FOR i := 0 TO (_Count - 1) DO
	IF _Data[i] = Item THEN
		_Data[i]	 := 0;
		removedItems := removedItems + 1;
	END_IF
END_FOR

IF _Count > 1 THEN
	FOR i := 0 TO (_Count - 2) DO
		IF _Data[i] = 0 AND _Data[i + 1] <> 0 THEN
			_Data[i]	 := _Data[i + 1];
			_Data[i + 1] := 0;
		END_IF
	END_FOR
END_IF

CountListItems();
_Count := _Count - removedItems;
END_METHOD

END_FUNCTION_BLOCK

// ---- _Internal/MotionTasks/MC2/AX5000/Mc2MotionTask_AX5000AmpToNm.TcPOU
FUNCTION_BLOCK Mc2MotionTask_AX5000AmpToNm EXTENDS Mc2MotionTask
VAR
	i					   : INT;
	SequenceState		   : DINT := -10;
	RawConfigChPeakCurrent : UDINT;					// Configured Channel Peak Current  ( raw )
	ConfigChPeakCurrent	   : LREAL;					// Configured Channel Peak Current  ( units := A )
	MotorConsType		   : WORD;					// Motor construction type          ( raw )
	MotorType			   : BOOL;					// Motor construction type          ( units := 0 = Rotary, 1 = Linear ) 
	RawContStallTorque	   : UDINT;					// Motor continuous stall torque    ( raw )
	ContStallTorque		   : LREAL;					// Motor continuous stall torque    ( units := Nm )
	ContStallTorqueEx	   : LREAL;					// Motor continuous stall torque    ( units := Nm ) - extended slope   
	RawPeakTorque		   : UDINT;					// Motor peak torque                ( raw )
	PeakTorque			   : LREAL;					// Motor peak torque                ( units := Nm )
	RawContStallForce	   : UDINT;					// Motor continuous stall force     ( raw )
	ContStallForce		   : LREAL;					// Motor continuous stall force     ( units := N )
	ContStallForceEx	   : LREAL;					// Motor continuous stall force     ( units := N ) - extended slope
	RawPeakForce		   : UDINT;					// Motor peak force                 ( raw )
	PeakForce			   : LREAL;					// Motor peak force                 ( units := N )
	RawContStallCurrent	   : UDINT;					// Motor continuous stall current   ( raw )
	ContStallCurrent	   : LREAL;					// Motor continuous stall current   ( units := A )
	ContStallCurrentEx	   : LREAL;					// Motor continuous stall current   ( units := A ) - extended slope
	RawPeakCurrent		   : UDINT;					// Motor peak current               ( raw )
	PeakCurrent			   : LREAL;					// Motor peak current               ( units := A )
	Scale				   : LREAL;					// Position between array indexes   ( units := % )
	SoERead				   : FB_SoERead;			// Read SoE params from drive
	RawMotorTorqueCurve	   : ST_IDN_P_0_0074_UDINT; // Contents read in from P-0-0074   ( raw )
END_VAR

VAR
	_ErrorId		 : UDINT;			 // 1 = Axis Not Linked, 2 = Failed To Read P-0-0074, 3 = Failed To Read P-0-0092, 4 = Failed To Read P-0-0050, 5 = Failed To Read P-0-0070, 6 = Failed To Read P-0-0126, 7 = Failed To Read S-0-0111
	CalculatedValues : ST_AX5000AmpToNm; // Data read in and calculated from the drive
END_VAR

(*  
Error Ids:
  1 = Axis Not Linked, 
  2 = Failed To Read P-0-0074,
  3 = Failed To Read P-0-0092, 
  4 = Failed To Read P-0-0050, 
  5 = Failed To Read P-0-0070, 
  6 = Failed To Read P-0-0126, 
  7 = Failed To Read S-0-0111 
*)

{attribute 'monitoring' := 'call'}
PROPERTY ActCurrent : LREAL
GET
ActCurrent := CalculatedValues.ActCurrent;
END_GET
END_PROPERTY

{attribute 'monitoring' := 'call'}
PROPERTY ActTorque : LREAL
GET
ActTorque := CalculatedValues.ActTorque;
END_GET
END_PROPERTY

{attribute 'monitoring' := 'call'}
PROPERTY Busy : BOOL
GET
Busy := SequenceState > 0 AND SequenceState <= 100;
END_GET
END_PROPERTY

METHOD CyclicLogic
IF _Axis = 0 THEN
	RETURN;
END_IF

CASE SequenceState OF
	-10: // Initialize
		RawConfigChPeakCurrent := 0;
		ConfigChPeakCurrent	   := 0.0;
		MotorConsType		   := 0;
		MotorType			   := FALSE;
		RawContStallTorque	   := 0;
		ContStallTorque		   := 0.0;
		ContStallTorqueEx	   := 0.0;
		RawPeakTorque		   := 0;
		PeakTorque			   := 0.0;
		RawContStallForce	   := 0;
		ContStallForce		   := 0.0;
		ContStallForceEx	   := 0.0;
		RawPeakForce		   := 0;
		PeakForce			   := 0.0;
		RawContStallCurrent	   := 0;
		ContStallCurrent	   := 0.0;
		ContStallCurrentEx	   := 0.0;
		RawPeakCurrent		   := 0;
		PeakCurrent			   := 0.0;
		Scale				   := 0.0;
		SoERead(Execute := FALSE, Axis := _Axis.Axis);
		MEMSET(ADR(RawMotorTorqueCurve), 16#0, SIZEOF(RawMotorTorqueCurve));
		MEMSET(ADR(CalculatedValues), 16#0, SIZEOF(CalculatedValues));
		IF _Axis.Axis.NcToPlc.AxisId = 0 THEN
			_ErrorId	  := 1;
			SequenceState := 5000;
		ELSE
			SequenceState := SequenceState + 10;
		END_IF

	0:	// Wait for Execute()  
	10: // Read in the value of P-0-0074 ( Motor torque characteristic )
		SoERead(NetId	:= '',
				Idn		:= P_0_IDNs + 74,
				Element := 16#40,
				pDstBuf := ADR(RawMotorTorqueCurve),
				BufLen	:= SIZEOF(RawMotorTorqueCurve),
				Execute := TRUE,
				Axis	:= _Axis.Axis);

		IF NOT SoERead.Busy AND NOT SoERead.Error THEN
			SoERead(Execute := FALSE, Axis := _Axis.Axis);
			FOR i := 0 TO 9 DO // Convert raw values into actual units
				CalculatedValues.Curve.Iq[i] := UDINT_TO_LREAL(RawMotorTorqueCurve.Elements.Iq[i]) / 1000.0;
				CalculatedValues.Curve.M[i]	 := UDINT_TO_LREAL(RawMotorTorqueCurve.Elements.M[i]) / 100.0;
			END_FOR

			SequenceState := SequenceState + 10;
		ELSIF SoERead.Error THEN
			SoERead(Execute := FALSE, Axis := _Axis.Axis);
			_ErrorId	  := 2;
			SequenceState := 5000;
		END_IF

	20: // Read in the value of P-0-0092 ( Configured channel peak current )       
		SoERead(NetId	:= '',
				Idn		:= P_0_IDNs + 92,
				Element := 16#40,
				pDstBuf := ADR(RawConfigChPeakCurrent),
				BufLen	:= SIZEOF(RawConfigChPeakCurrent),
				Execute := TRUE,
				Axis	:= _Axis.Axis);

		IF NOT SoERead.Busy AND NOT SoERead.Error THEN // Convert raw values into actual units
			SoERead(Execute := FALSE, Axis := _Axis.Axis);
			ConfigChPeakCurrent := UDINT_TO_LREAL(RawConfigChPeakCurrent) / 1000.0;
			SequenceState		:= SequenceState + 10;
		ELSIF SoERead.Error THEN
			SoERead(Execute := FALSE, Axis := _Axis.Axis);
			_ErrorId	  := 3;
			SequenceState := 5000;
		END_IF

	30: // Check for valid characteristic curve
		IF RawMotorTorqueCurve.Elements.Iq[9] = 0 THEN
			SequenceState := SequenceState + 10; // Curve is not available
		ELSE
			SequenceState := 1000; // Curve is available
		END_IF

	40: // Read in the value of P-0-0050 ( Motor construction type )       
		SoERead(NetId	:= '',
				Idn		:= P_0_IDNs + 50,
				Element := 16#40,
				pDstBuf := ADR(MotorConsType),
				BufLen	:= SIZEOF(MotorConsType),
				Execute := TRUE,
				Axis	:= _Axis.Axis);

		IF NOT SoERead.Busy AND NOT SoERead.Error THEN
			SoERead(Execute := FALSE, Axis := _Axis.Axis);
			MotorType := MotorConsType.1;
			IF NOT MotorType THEN
				SequenceState := 50; // Rotary
			ELSE
				SequenceState := 70; // Linear
			END_IF
		ELSIF SoERead.Error THEN
			SoERead(Execute := FALSE, Axis := _Axis.Axis);
			_ErrorId	  := 4;
			SequenceState := 5000;
		END_IF

	50: // Read in the value of P-0-0070 ( Motor continuous stall torque )       
		SoERead(NetId	:= '',
				Idn		:= P_0_IDNs + 70,
				Element := 16#40,
				pDstBuf := ADR(RawContStallTorque),
				BufLen	:= SIZEOF(RawContStallTorque),
				Execute := TRUE,
				Axis	:= _Axis.Axis);

		IF NOT SoERead.Busy AND NOT SoERead.Error THEN
			SoERead(Execute := FALSE, Axis := _Axis.Axis);
			ContStallTorque := UDINT_TO_LREAL(RawContStallTorque) / 100.0;
			SequenceState	:= SequenceState + 10;
		ELSIF SoERead.Error THEN
			SoERead(Execute := FALSE, Axis := _Axis.Axis);
			_ErrorId	  := 5;
			SequenceState := 5000;
		END_IF

	60: // Read in the value of P-0-0073 ( Motor peak torque )       
		SoERead(NetId	:= '',
				Idn		:= P_0_IDNs + 73,
				Element := 16#40,
				pDstBuf := ADR(RawPeakTorque),
				BufLen	:= SIZEOF(RawPeakTorque),
				Execute := TRUE,
				Axis	:= _Axis.Axis);

		IF NOT SoERead.Busy AND NOT SoERead.Error THEN
			SoERead(Execute := FALSE, Axis := _Axis.Axis);
			PeakTorque	  := UDINT_TO_LREAL(RawPeakTorque) / 100.0;
			SequenceState := 90;
		ELSIF SoERead.Error THEN
			SoERead(Execute := FALSE, Axis := _Axis.Axis);
			SequenceState := 90;
		END_IF

	70: // Read in the value of P-0-0126 ( Motor continuous stall force )       
		SoERead(NetId	:= '',
				Idn		:= P_0_IDNs + 126,
				Element := 16#40,
				pDstBuf := ADR(RawContStallForce),
				BufLen	:= SIZEOF(RawContStallForce),
				Execute := TRUE,
				Axis	:= _Axis.Axis);

		IF NOT SoERead.Busy AND NOT SoERead.Error THEN
			SoERead(Execute := FALSE, Axis := _Axis.Axis);
			ContStallForce := UDINT_TO_LREAL(RawContStallForce) / 100.0;
			SequenceState  := SequenceState + 10;
		ELSIF SoERead.Error THEN
			SoERead(Execute := FALSE, Axis := _Axis.Axis);
			_ErrorId	  := 6;
			SequenceState := 5000;
		END_IF

	80: // Read in the value of P-0-0128 ( Motor peak force )       
		SoERead(NetId	:= '',
				Idn		:= P_0_IDNs + 128,
				Element := 16#40,
				pDstBuf := ADR(RawPeakForce),
				BufLen	:= SIZEOF(RawPeakForce),
				Execute := TRUE,
				Axis	:= _Axis.Axis);

		IF NOT SoERead.Busy AND NOT SoERead.Error THEN
			SoERead(Execute := FALSE, Axis := _Axis.Axis);
			PeakForce	  := UDINT_TO_LREAL(RawPeakForce) / 100.0;
			SequenceState := SequenceState + 10;
		ELSIF SoERead.Error THEN
			SoERead(Execute := FALSE, Axis := _Axis.Axis);
			SequenceState := SequenceState + 10;
		END_IF

	90: // Read in the value of S-0-0111 ( Motor continuous stall current )       
		SoERead(NetId	:= '',
				Idn		:= S_0_IDNs + 111,
				Element := 16#40,
				pDstBuf := ADR(RawContStallCurrent),
				BufLen	:= SIZEOF(RawContStallCurrent),
				Execute := TRUE,
				Axis	:= _Axis.Axis);

		IF NOT SoERead.Busy AND NOT SoERead.Error THEN
			SoERead(Execute := FALSE, Axis := _Axis.Axis);
			ContStallCurrent := UDINT_TO_LREAL(RawContStallCurrent) / 1000.0;
			SequenceState	 := SequenceState + 10;
		ELSIF SoERead.Error THEN
			SoERead(Execute := FALSE, Axis := _Axis.Axis);
			_ErrorId	  := 7;
			SequenceState := 5000;
		END_IF

	100: // Read in the value of S-0-0109 ( Motor peak current )       
		SoERead(NetId	:= '',
				Idn		:= S_0_IDNs + 109,
				Element := 16#40,
				pDstBuf := ADR(RawPeakCurrent),
				BufLen	:= SIZEOF(RawPeakCurrent),
				Execute := TRUE,
				Axis	:= _Axis.Axis);

		IF NOT SoERead.Busy THEN
			SoERead(Execute := FALSE, Axis := _Axis.Axis);
			PeakCurrent := UDINT_TO_LREAL(RawPeakCurrent) / 1000.0;
			IF NOT MotorType THEN
				IF PeakCurrent = 0 OR PeakTorque = 0 THEN
					SequenceState := 300; // Rotary Motor: Curve not available... peak torque and current missing - Using slope of points 0,0 to P-0-0070 and S-0-0111
				ELSE
					SequenceState := 200; // Rotary Motor: Curve not available - Using linear interpolation of points P-0-0070, P-0-0073, S-0-0111 and S-0-0109
				END_IF
			ELSE
				IF PeakCurrent = 0 OR PeakForce = 0 THEN
					SequenceState := 500; // Linear Motor: Curve not available... peak torque and current missing - Using slope of points 0,0 to P-0-0126 and S-0-0111
				ELSE
					SequenceState := 400; // Linear Motor: Curve not available - Using linear interpolation of points P-0-0126, P-0-0128, S-0-0111 and S-0-0109
				END_IF
			END_IF
		END_IF

	200: // Rotary Motor: Curve not available - Using linear interpolation of points P-0-0070, P-0-0073, S-0-0111 and S-0-0109
		CalculatedValues.ActCurrent := ABS((_Axis.Axis.NcToPlc.ActTorque / 100) * ConfigChPeakCurrent);
		// Convert the actual current in amps to Nm
		IF CalculatedValues.ActCurrent = 0 THEN
			CalculatedValues.ActTorque := 0;
		ELSIF CalculatedValues.ActCurrent > 0 AND CalculatedValues.ActCurrent < ContStallCurrent THEN
			IF ContStallCurrent > 0 THEN
				Scale					   := CalculatedValues.ActCurrent / ContStallCurrent;
				CalculatedValues.ActTorque := Scale * ContStallTorque;
			END_IF
		ELSIF CalculatedValues.ActCurrent >= ContStallCurrent AND CalculatedValues.ActCurrent <= PeakCurrent THEN
			IF (CalculatedValues.ActCurrent - ContStallCurrent) > 0 AND (PeakCurrent - ContStallCurrent) > 0 THEN
				Scale					   := (CalculatedValues.ActCurrent - ContStallCurrent) / (PeakCurrent - ContStallCurrent);
				CalculatedValues.ActTorque := (Scale * (PeakTorque - ContStallTorque) + ContStallTorque);
			END_IF
		END_IF

	300: // Rotary Motor: Curve not available... peak torque and current missing - Using slope of points 0,0 to P-0-0070 and S-0-0111
		CalculatedValues.ActCurrent := ABS((_Axis.Axis.NcToPlc.ActTorque / 100) * ConfigChPeakCurrent);

		// Project slope from continuous stall torque/current
		ContStallCurrentEx := ContStallCurrent * 10.0;
		ContStallTorqueEx  := ContStallTorque * 10.0;
		// Convert the actual current in amps to Nm
		IF CalculatedValues.ActCurrent = 0 THEN
			CalculatedValues.ActTorque := 0;
		ELSIF CalculatedValues.ActCurrent > 0 AND CalculatedValues.ActCurrent <= ContStallCurrentEx THEN
			IF ContStallCurrentEx > 0 THEN
				Scale					   := CalculatedValues.ActCurrent / ContStallCurrentEx;
				CalculatedValues.ActTorque := Scale * ContStallTorqueEx;
			END_IF
		END_IF

	400: // Linear Motor: Curve not available - Using linear interpolation of points P-0-0126, P-0-0128, S-0-0111 and S-0-0109
		CalculatedValues.ActCurrent := ABS((_Axis.Axis.NcToPlc.ActTorque / 100) * ConfigChPeakCurrent);
		// Convert the actual current in amps to Nm
		IF CalculatedValues.ActCurrent = 0 THEN
			CalculatedValues.ActTorque := 0;
		ELSIF CalculatedValues.ActCurrent > 0 AND CalculatedValues.ActCurrent < ContStallCurrent THEN
			IF ContStallCurrent > 0 THEN
				Scale					   := CalculatedValues.ActCurrent / ContStallCurrent;
				CalculatedValues.ActTorque := Scale * ContStallForce;
			END_IF
		ELSIF CalculatedValues.ActCurrent >= ContStallCurrent AND CalculatedValues.ActCurrent <= PeakCurrent THEN
			IF (CalculatedValues.ActCurrent - ContStallCurrent) > 0 AND (PeakCurrent - ContStallCurrent) > 0 THEN
				Scale					   := (CalculatedValues.ActCurrent - ContStallCurrent) / (PeakCurrent - ContStallCurrent);
				CalculatedValues.ActTorque := (Scale * (PeakForce - ContStallForce) + ContStallForce);
			END_IF
		END_IF

	500: // Linear Motor: Curve not available... peak torque and current missing - Using slope of points 0,0 to P-0-0126 and S-0-0111
		CalculatedValues.ActCurrent := ABS((_Axis.Axis.NcToPlc.ActTorque / 100) * ConfigChPeakCurrent);

		// Project slope from continuous stall torque/current
		ContStallCurrentEx := ContStallCurrent * 10.0;
		ContStallForceEx   := ContStallForce * 10.0;
		// Convert the actual current in amps to Nm
		IF CalculatedValues.ActCurrent = 0 THEN
			CalculatedValues.ActTorque := 0;
		ELSIF CalculatedValues.ActCurrent > 0 AND CalculatedValues.ActCurrent <= ContStallCurrentEx THEN
			IF ContStallCurrentEx > 0 THEN
				Scale					   := CalculatedValues.ActCurrent / ContStallCurrentEx;
				CalculatedValues.ActTorque := Scale * ContStallForceEx;
			END_IF
		END_IF

	1000: // Rotary or Linear Motor: Curve available - Compare actual torque value in Amps to the characteristic curve and output actual torque value in Nm
		CalculatedValues.ActCurrent := ABS((_Axis.Axis.NcToPlc.ActTorque / 100) * ConfigChPeakCurrent);
		// Convert the actual current in amps to Nm
		FOR i := 1 TO 9 DO
			IF CalculatedValues.ActCurrent = 0 THEN
				CalculatedValues.ActTorque := 0;
				EXIT;
			ELSIF CalculatedValues.ActCurrent > 0 AND CalculatedValues.ActCurrent < CalculatedValues.Curve.Iq[0] THEN
				IF CalculatedValues.Curve.Iq[0] > 0 THEN
					Scale					   := CalculatedValues.ActCurrent / CalculatedValues.Curve.Iq[0];
					CalculatedValues.ActTorque := Scale * CalculatedValues.Curve.M[0];
				END_IF

				EXIT;
			ELSIF CalculatedValues.ActCurrent >= CalculatedValues.Curve.Iq[i - 1] AND CalculatedValues.ActCurrent <= CalculatedValues.Curve.Iq[i] THEN
				IF (CalculatedValues.Curve.Iq[i] - CalculatedValues.Curve.Iq[i - 1]) > 0 AND CalculatedValues.ActCurrent - CalculatedValues.Curve.Iq[i - 1] > 0 THEN
					Scale					   := (CalculatedValues.ActCurrent - CalculatedValues.Curve.Iq[i - 1]) / (CalculatedValues.Curve.Iq[i] - CalculatedValues.Curve.Iq[i - 1]);
					CalculatedValues.ActTorque := (Scale * (CalculatedValues.Curve.M[i] - CalculatedValues.Curve.M[i - 1]) + CalculatedValues.Curve.M[i - 1]);
				END_IF

				EXIT;
			END_IF
		END_FOR

	5000: // Error state        
		SequenceState := -10;
END_CASE
END_METHOD

{attribute 'monitoring' := 'call'}
PROPERTY Error : BOOL
GET
Error := SequenceState = 5000;
END_GET
END_PROPERTY

{attribute 'monitoring' := 'call'}
PROPERTY ErrorId : UDINT
GET
ErrorId := _ErrorId;
END_GET
END_PROPERTY

METHOD Execute : BOOL
IF Busy THEN
	RETURN;
END_IF

SequenceState := 10;
_ErrorID	  := 0;
Execute		  := TRUE;
END_METHOD

END_FUNCTION_BLOCK

// ---- _Internal/MotionTasks/MC2/Home/Mc2MotionHomeTask_CoESetEncoderOffset.TcPOU
FUNCTION_BLOCK Mc2MotionHomeTask_CoESetEncoderOffset EXTENDS Mc2MotionTask
VAR
	SequenceState	  : UDINT;
	SetPositionOffset : FB_CoEAX8000SetPositionOffset;
	_HomePosition	  : LREAL := 0.0;
	_ErrorId		  : UDINT;
END_VAR

{attribute 'monitoring' := 'call'}
PROPERTY Busy : BOOL
GET
Busy := SequenceState <> 0;
END_GET
END_PROPERTY

METHOD CyclicLogic
VAR_INST
	DriveEnabledAtBeginning : BOOL;
	AxisRef					: REFERENCE TO Tc2_MC2.AXIS_REF;
END_VAR
CASE SequenceState OF
	0: // Wait for Execute();
	10:
		IF Axis.Enabled THEN
			DriveEnabledAtBeginning := TRUE;
			SequenceState			:= 20;
		ELSE
			DriveEnabledAtBeginning := FALSE;
			SequenceState			:= 30;
		END_IF

	20:
		Axis.Disable();
		IF NOT Axis.Enabled THEN
			SequenceState := 30;
		END_IF

	30:
		AxisRef REF= Axis.Axis;
		SetPositionOffset(Axis	   := AxisRef,
						  Execute  := TRUE,
						  Position := _HomePosition,
						  Relative := FALSE,
						  Feedback := ePositionOffsetFeedback1,
						  Memory   := ePositionOffsetMemory_Encoder);

		IF NOT SetPositionOffset.Busy THEN
			IF SetPositionOffset.Error THEN
				_ErrorId	  := SetPositionOffset.ErrorID;
				SequenceState := 999;
			ELSE
				SequenceState := 40;
			END_IF

			SetPositionOffset(Axis := AxisRef, Execute := FALSE);
		END_IF

	40:
		IF DriveEnabledAtBeginning THEN
			SequenceState := 50;
		ELSE
			SequenceState := 0;
		END_IF

	50:
		Axis.Enable();
		IF Axis.Enabled THEN
			SequenceState := 0;
		END_IF

	999:
		_ErrorId	  := 0;
		SequenceState := 0;
END_CASE
END_METHOD

{attribute 'monitoring' := 'call'}
PROPERTY Error : BOOL
GET
Error := SequenceState = 999;
END_GET
END_PROPERTY

{attribute 'monitoring' := 'call'}
PROPERTY ErrorId : UDINT
GET
ErrorId := _ErrorId;
END_GET
END_PROPERTY

METHOD Execute : BOOL
IF Axis.Busy OR Axis.Error THEN
	RETURN;
END_IF

SequenceState := 10;
_ErrorID	  := 0;
Execute		  := TRUE;
END_METHOD

{attribute 'monitoring' := 'call'}
PROPERTY HomePosition : LREAL
GET
HomePosition := _HomePosition;
END_GET
SET
_HomePosition := HomePosition;
END_SET
END_PROPERTY

END_FUNCTION_BLOCK

// ---- _Internal/MotionTasks/MC2/Home/Mc2MotionHomeTask_SetPosition.TcPOU
FUNCTION_BLOCK Mc2MotionHomeTask_SetPosition EXTENDS Mc2MotionTask
VAR
	MCSetPosition : Tc2_MC2.MC_SetPosition;
	_HomePosition : LREAL := 0.0;
END_VAR

{attribute 'monitoring' := 'call'}
PROPERTY Busy : BOOL
GET
Busy := MCSetPosition.Busy;
END_GET
END_PROPERTY

METHOD CyclicLogic
MCSetPosition(Axis := _Axis.Axis, Position := HomePosition);
MCSetPosition.Execute := FALSE;
END_METHOD

{attribute 'monitoring' := 'call'}
PROPERTY Error : BOOL
GET
Error := MCSetPosition.Error;
END_GET
END_PROPERTY

{attribute 'monitoring' := 'call'}
PROPERTY ErrorId : UDINT
GET
ErrorId := MCSetPosition.ErrorID;
END_GET
END_PROPERTY

METHOD Execute : BOOL
IF Axis.Busy OR Axis.Error THEN
	RETURN;
END_IF

MCSetPosition.Execute := TRUE;
Execute				  := TRUE;
END_METHOD

PROPERTY HomePosition : LREAL
GET
HomePosition := MCSetPosition.Position;
END_GET
SET
MCSetPosition.Position := HomePosition;
END_SET
END_PROPERTY

END_FUNCTION_BLOCK

// ---- _Internal/MotionTasks/MC2/Home/Mc2MotionHomeTask_SetPositionOffset.TcPOU
FUNCTION_BLOCK Mc2MotionHomeTask_SetPositionOffset EXTENDS Mc2MotionTask
VAR
	SequenceState	  : UDINT;
	SetPositionOffset : Tc2_MC2_Drive.FB_SetPositionOffset;
	_HomePosition	  : LREAL := 0.0;
	_ErrorId		  : UDINT;
	_Feedback		  : Tc2_MC2_Drive.E_PositionOffsetFeedback := Tc2_MC2_Drive.E_PositionOffsetFeedback.ePositionOffsetFeedback1;
	_Memory			  : Tc2_MC2_Drive.E_PositionOffsetMemory   := Tc2_MC2_Drive.E_PositionOffsetMemory.ePositionOffsetMemory_Encoder;
END_VAR

{attribute 'monitoring' := 'call'}
PROPERTY Busy : BOOL
GET
Busy := SequenceState <> 0;
END_GET
END_PROPERTY

METHOD CyclicLogic
VAR_INST
	DriveEnabledAtBeginning : BOOL;
	AxisRef					: REFERENCE TO Tc2_MC2.AXIS_REF;
END_VAR
CASE SequenceState OF
	0: // Wait for Execute();
	10:
		IF Axis.Enabled THEN
			DriveEnabledAtBeginning := TRUE;
			SequenceState			:= 20;
		ELSE
			DriveEnabledAtBeginning := FALSE;
			SequenceState			:= 30;
		END_IF

	20:
		Axis.Disable();
		IF NOT Axis.Enabled THEN
			SequenceState := 30;
		END_IF

	30:
		AxisRef REF= Axis.Axis;
		SetPositionOffset(Axis	   := AxisRef,
						  Execute  := TRUE,
						  Position := _HomePosition,
						  Relative := FALSE,
						  Feedback := _Feedback,
						  Memory   := _Memory);

		IF NOT SetPositionOffset.Busy THEN
			IF SetPositionOffset.Error THEN
				_ErrorId	  := SetPositionOffset.ErrorID;
				SequenceState := 999;
			ELSE
				SequenceState := 40;
			END_IF

			SetPositionOffset(Axis := AxisRef, Execute := FALSE);
		END_IF

	40:
		IF DriveEnabledAtBeginning THEN
			SequenceState := 50;
		ELSE
			SequenceState := 0;
		END_IF

	50:
		Axis.Enable();
		IF Axis.Enabled THEN
			SequenceState := 0;
		END_IF

	999:
		_ErrorId	  := 0;
		SequenceState := 0;
END_CASE
END_METHOD

{attribute 'monitoring' := 'call'}
PROPERTY Error : BOOL
GET
Error := SequenceState = 999;
END_GET
END_PROPERTY

{attribute 'monitoring' := 'call'}
PROPERTY ErrorId : UDINT
GET
ErrorId := _ErrorId;
END_GET
END_PROPERTY

METHOD Execute : BOOL
IF Axis.Busy OR Axis.Error THEN
	RETURN;
END_IF

SequenceState := 10;
_ErrorID	  := 0;
Execute		  := TRUE;
END_METHOD

{attribute 'monitoring' := 'call'}
PROPERTY Feedback : E_PositionOffsetFeedback
SET
_Feedback := Feedback;
END_SET
END_PROPERTY

{attribute 'monitoring' := 'call'}
PROPERTY HomePosition : LREAL
GET
HomePosition := _HomePosition;
END_GET
SET
_HomePosition := HomePosition;
END_SET
END_PROPERTY

{attribute 'monitoring' := 'call'}
PROPERTY Memory : E_PositionOffsetMemory
SET
_Memory := Memory;
END_SET
END_PROPERTY

END_FUNCTION_BLOCK

// ---- _Internal/MotionTasks/MC2/Home/Mc2MotionHomeTask_SetZeroHere.TcPOU
FUNCTION_BLOCK Mc2MotionHomeTask_SetZeroHere EXTENDS Mc2MotionTask
VAR
	MCSetPosition : Tc2_MC2.MC_SetPosition;
END_VAR

{attribute 'monitoring' := 'call'}
PROPERTY Busy : BOOL
GET
Busy := MCSetPosition.Busy;
END_GET
END_PROPERTY

METHOD CyclicLogic
MCSetPosition(Axis := _Axis.Axis);
MCSetPosition.Execute := FALSE;
END_METHOD

{attribute 'monitoring' := 'call'}
PROPERTY Error : BOOL
GET
Error := MCSetPosition.Error;
END_GET
END_PROPERTY

{attribute 'monitoring' := 'call'}
PROPERTY ErrorId : UDINT
GET
ErrorId := MCSetPosition.ErrorID;
END_GET
END_PROPERTY

METHOD Execute : BOOL
IF Axis.Busy OR Axis.Error THEN
	RETURN;
END_IF

MCSetPosition.Execute := TRUE;
Execute				  := TRUE;
END_METHOD

END_FUNCTION_BLOCK

// ---- _Internal/MotionTasks/MC2/Home/Mc2MotionHomeTask_TouchProbe.TcPOU
FUNCTION_BLOCK Mc2MotionHomeTask_TouchProbe EXTENDS Mc2MotionTask
VAR
	InputState AT %I*	 : BOOL;
	SequenceState		 : UDINT;
	MCStepAbsoluteSwitch : MC_StepAbsoluteSwitchDetection;
	MCFinishHoming		 : MC_FinishHoming;
	MCAbortHoming		 : MC_AbortHoming;
	HomingParameters	 : MC_HomingParameter;
	SignalRef			 : MC_Ref_Signal_Ref := (SignalSource := E_SignalSource.SignalSource_Default, TouchProbe := E_TouchProbe.PlcEvent);
	SetPositionOffset	 : FB_SetPositionOffset;
	MCMoveRelative		 : Tc2_MC2.MC_MoveRelative;
	SensorPosition		 : LREAL;
	NewFinalPosition	 : LREAL;
	_ErrorId			 : UDINT;
	_HomePosition		 : LREAL := 0.0;
	_TorqueLimit		 : LREAL := 40.0;
	_Velocity			 : LREAL := 20.0;
END_VAR

VAR CONSTANT
	IDLE_STATE	: UDINT := 0;
	ERROR_STATE : UDINT := 999;
END_VAR

{attribute 'monitoring' := 'call'}
PROPERTY Busy : BOOL
GET
Busy := SequenceState <> IDLE_STATE AND SequenceState <> ERROR_STATE;
END_GET
END_PROPERTY

METHOD CyclicLogic
VAR_INST
	ipEnablable : I_Enablable;
END_VAR
IF _Axis <> 0 THEN
    SignalRef.Level := InputState;
	CASE SequenceState OF
		10:
			IF NOT __QUERYINTERFACE(Axis, ipEnablable) THEN
				_ErrorId	  := E_AdsErr.DEVICE_SRVNOTSUPP;
				SequenceState := ERROR_STATE;
			ELSE
				NextMinorStep(SequenceState);
			END_IF

		11:
			IF NOT ipEnablable.Enabled THEN
				SequenceState := ERROR_STATE;
			ELSE
				NextMinorStep(SequenceState);
			END_IF

		12:
			IF InputState THEN
				NextMinorStep(SequenceState);
			ELSE
				NextStep(SequenceState);
			END_IF

		13:
			MCMoveRelative(Axis		:= _Axis.Axis,
						   Execute	:= TRUE,
						   Distance := 25.0,
						   Velocity := _Velocity);

			IF NOT MCMoveRelative.Busy THEN
				IF MCMoveRelative.Error THEN
					_ErrorId	  := MCMoveRelative.ErrorID;
					SequenceState := ERROR_STATE;
				ELSIF MCMoveRelative.Done THEN
					NextStep(SequenceState);
				END_IF

				MCMoveRelative(Axis := _Axis.Axis, Execute := FALSE);
			END_IF

		20:
			MCStepAbsoluteSwitch(Axis			 := _Axis.Axis,
								 Parameter		 := HomingParameters,
								 Execute		 := TRUE,
								 Direction		 := MC_Home_Direction.mcSwitchNegative,
								 SwitchMode		 := MC_Switch_Mode.mcEdgeSwitchNegative,
								 ReferenceSignal := SignalRef,
								 Velocity		 := _Velocity,
								 TimeLimit		 := TO_TIME((540.0 / _Velocity) * 1000.0),
								 TorqueLimit	 := _TorqueLimit);

			IF NOT MCStepAbsoluteSwitch.Busy THEN
				IF MCStepAbsoluteSwitch.Error THEN
					_ErrorId	  := MCStepAbsoluteSwitch.ErrorID;
					SequenceState := ERROR_STATE;
				ELSIF MCStepAbsoluteSwitch.Done THEN
					SensorPosition := MCStepAbsoluteSwitch.RecordedPosition;
					NextMinorStep(SequenceState);
				END_IF

				MCStepAbsoluteSwitch(Axis := _Axis.Axis, Parameter := HomingParameters, Execute := FALSE);
			END_IF

		21:
			IF _Axis.Axis.NcToPlc.SetVelo = 0.0 THEN
				NewFinalPosition := (_Axis.Axis.NcToPlc.SetPos - SensorPosition) + _HomePosition;
				NextStep(SequenceState);
			END_IF

		30:
			ipEnablable.Disable();
			IF NOT ipEnablable.Enabled THEN
				NextMinorStep(SequenceState);
			END_IF

		31:
			SetPositionOffset(Axis	   := _Axis.Axis,
							  Execute  := TRUE,
							  Position := NewFinalPosition,
							  Relative := FALSE,
							  Feedback := ePositionOffsetFeedback1,
							  Memory   := ePositionOffsetMemory_Drive);

			IF NOT SetPositionOffset.Busy THEN
				IF SetPositionOffset.Error THEN
					_ErrorId	  := SetPositionOffset.ErrorID;
					SequenceState := ERROR_STATE;
				ELSE
					NextStep(SequenceState);
				END_IF

				SetPositionOffset(Axis := _Axis.Axis, Execute := FALSE);
			END_IF

		40:
			ipEnablable.Enable();
			IF ipEnablable.Enabled THEN
				NextMinorStep(SequenceState);
			END_IF

		41:
			MCFinishHoming(Axis		 := _Axis.Axis,
						   Parameter := HomingParameters,
						   Execute	 := TRUE,
						   Distance	 := _Axis.Axis.NcToPlc.SetPos * -1.0,
						   Velocity	 := _Velocity);

			IF NOT MCFinishHoming.Busy THEN
				IF MCFinishHoming.Error THEN
					_ErrorId	  := MCFinishHoming.ErrorID;
					SequenceState := ERROR_STATE;
				ELSE
					SequenceState := IDLE_STATE;
				END_IF

				MCFinishHoming(Axis := _Axis.Axis, Parameter := HomingParameters, Execute := FALSE);
			END_IF

		ERROR_STATE:
			MCAbortHoming(Axis := _Axis.Axis, Parameter := HomingParameters, Execute := TRUE);
	END_CASE
END_IF
END_METHOD

{attribute 'monitoring' := 'call'}
PROPERTY Error : BOOL
GET
Error := SequenceState = ERROR_STATE;
END_GET
END_PROPERTY

{attribute 'monitoring' := 'call'}
PROPERTY ErrorId : UDINT
GET
ErrorId := _ErrorId;
END_GET
END_PROPERTY

METHOD Execute : BOOL
IF (_Axis = 0) OR Busy THEN
	RETURN;
END_IF

MCAbortHoming(Axis := _Axis.Axis, Parameter := HomingParameters, Execute := FALSE);
SequenceState := 10;
_ErrorID	  := 0;
Execute		  := TRUE;
END_METHOD

PROPERTY HomePosition : LREAL
GET
HomePosition := _HomePosition;
END_GET
SET
_HomePosition := HomePosition;
END_SET
END_PROPERTY

PROPERTY TorqueLimit : LREAL
GET
TorqueLimit := _TorqueLimit;
END_GET
SET
_TorqueLimit := TorqueLimit;
END_SET
END_PROPERTY

PROPERTY Velocity : LREAL
GET
Velocity := _Velocity;
END_GET
SET
_Velocity := Velocity;
END_SET
END_PROPERTY

END_FUNCTION_BLOCK

// ---- _Internal/MotionTasks/MC2/Power/Mc2StopTask.TcPOU
FUNCTION_BLOCK Mc2StopTask EXTENDS Mc2MotionTask IMPLEMENTS I_Mc2MotionTask
VAR
	McHalt		  : Tc2_MC2.MC_Halt;
	_McBufferMode : Tc2_MC2.MC_BufferMode;
	_MoveOptions  : Tc2_MC2.ST_MoveOptions;
END_VAR

PROPERTY BufferMode : REFERENCE TO MC_BufferMode
GET
BufferMode REF= _McBufferMode;
END_GET
END_PROPERTY

{attribute 'monitoring' := 'call'}
PROPERTY Busy : BOOL
GET
Busy := McHalt.Busy;
END_GET
END_PROPERTY

METHOD CyclicLogic
McHalt(Axis			:= _Axis.Axis,
	   Deceleration := _Axis.Deceleration,
	   Jerk			:= _Axis.Jerk,
	   BufferMode	:= _McBufferMode,
	   Options		:= _MoveOptions);

McHalt.Execute := FALSE;
END_METHOD

{attribute 'monitoring' := 'call'}
PROPERTY Error : BOOL
GET
Error := McHalt.Error;
END_GET
END_PROPERTY

{attribute 'monitoring' := 'call'}
PROPERTY ErrorId : UDINT
GET
ErrorId := McHalt.ErrorID;
END_GET
END_PROPERTY

METHOD Execute : BOOL
McHalt(Axis			:= _Axis.Axis,
	   Execute		:= TRUE,
	   Deceleration := _Axis.Deceleration,
	   Jerk			:= _Axis.Jerk,
	   BufferMode	:= _McBufferMode,
	   Options		:= _MoveOptions);

Execute := TRUE;
END_METHOD

PROPERTY MoveOptions : REFERENCE TO ST_MoveOptions
GET
MoveOptions REF= _MoveOptions;
END_GET
END_PROPERTY

END_FUNCTION_BLOCK

// ---- _Internal/MotionTasks/MC2/Reset/Mc2CoEExtendedResetTask.TcPOU
FUNCTION_BLOCK Mc2CoEExtendedResetTask EXTENDS Mc2MotionTask
VAR
	DriveErrorCode AT %I* : UINT;
	CoERead				  : FB_CoERead;
	CoEWrite			  : FB_CoEWrite;
	MCReset				  : Tc2_MC2.MC_Reset;
	SequenceState		  : UDINT;
	_ErrorID			  : UDINT;
END_VAR

{attribute 'monitoring' := 'call'}
PROPERTY Busy : BOOL
GET
Busy := SequenceState <> 0;
END_GET
END_PROPERTY

METHOD CyclicLogic
VAR_INST
	AlwaysTrue			 : USINT := 1;
	ExtendedResetEnabled : BOOL;
END_VAR
CASE SequenceState OF
	0: // Wait for Execute()
	10:
		IF (_Axis.Axis.Status.DriveDeviceError) THEN
			IF NOT ExtendedResetEnabled THEN
				IF (DriveErrorCode = 16#8185) OR (DriveErrorCode = 16#63A0) THEN
					SequenceState := SequenceState + 10;
				ELSIF (DriveErrorCode = 16#63A2) OR (DriveErrorCode = 16#63A4) THEN
					SequenceState := 100;
				END_IF
			ELSE
				SequenceState := 100;
			END_IF
		ELSE
			ExtendedResetEnabled := FALSE;
		END_IF

	20:
		CoEWrite(Axis	  := _Axis.Axis,
				 Index	  := 16#3004,
				 SubIndex := 16#4,
				 pSrcBuf  := ADR(AlwaysTrue),
				 BufLen	  := SIZEOF(USINT),
				 Execute  := TRUE);

		IF NOT CoEWrite.Busy THEN
			IF CoEWrite.Error THEN
				IF CoEWrite.AdsErrId > 0 THEN
					_ErrorID := CoEWrite.AdsErrId;
				ELSE
					_ErrorID := CoEWrite.CANopenErrId;
				END_IF

				SequenceState := 999;
			ELSE
				SequenceState := SequenceState + 1;
			END_IF

			CoEWrite(Axis := _Axis.Axis, Execute := FALSE);
		END_IF

	21:
		CoEWrite(Axis	  := _Axis.Axis,
				 Index	  := 16#3404,
				 SubIndex := 16#4,
				 pSrcBuf  := ADR(AlwaysTrue),
				 BufLen	  := SIZEOF(USINT),
				 Execute  := TRUE);

		IF NOT CoEWrite.Busy THEN
			IF CoEWrite.Error THEN
				IF CoEWrite.AdsErrId > 0 THEN
					_ErrorID := CoEWrite.AdsErrId;
				ELSE
					_ErrorID := CoEWrite.CANopenErrId;
				END_IF

				SequenceState := 999;
			ELSE
				SequenceState := SequenceState + 1;
			END_IF

			CoEWrite(Axis := _Axis.Axis, Execute := FALSE);
		END_IF

	22:
		ExtendedResetEnabled := TRUE;
		SequenceState		 := 1000;

	100:
		MCReset.Execute := TRUE;
		SequenceState	:= SequenceState + 10;

	110:
		IF NOT MCReset.Busy THEN
			SequenceState := 0;
		END_IF

	999:
		_ErrorID	  := 0;
		SequenceState := 0;
END_CASE

MCReset(Axis := _Axis.Axis);
MCReset.Execute := FALSE;
END_METHOD

{attribute 'monitoring' := 'call'}
PROPERTY Error : BOOL
GET
Error := SequenceState = 999;
END_GET
END_PROPERTY

{attribute 'monitoring' := 'call'}
PROPERTY ErrorId : UDINT
GET
ErrorId := _ErrorID;
END_GET
END_PROPERTY

METHOD Execute : BOOL
IF _Axis.Axis.Status.Coupled AND NOT _Axis.Axis.Status.Error THEN
	Execute := TRUE;
	RETURN;
ELSIF Busy OR _Axis.Axis.Status.Coupled THEN
	Execute := TRUE;
	RETURN;
END_IF

SequenceState := 10;
Execute		  := TRUE;
END_METHOD

END_FUNCTION_BLOCK

// ---- _Internal/MotionTasks/MC2/Reset/Mc2CoEResetTask.TcPOU
FUNCTION_BLOCK Mc2CoEResetTask EXTENDS Mc2MotionTask
VAR
	MCReset		  : Tc2_MC2.MC_Reset;
	SequenceState : UDINT;
END_VAR

{attribute 'monitoring' := 'call'}
PROPERTY Busy : BOOL
GET
Busy := SequenceState <> 0;
END_GET
END_PROPERTY

METHOD CyclicLogic
CASE SequenceState OF
	0: // Wait for Execute()
	10:
		MCReset.Execute := TRUE;
		SequenceState	:= SequenceState + 10;

	20:
		IF NOT MCReset.Busy THEN
			SequenceState := 0;
		END_IF
END_CASE

MCReset(Axis := _Axis.Axis);
MCReset.Execute := FALSE;
END_METHOD

{attribute 'monitoring' := 'call'}
PROPERTY Error : BOOL
GET
Error := MCReset.Error;
END_GET
END_PROPERTY

{attribute 'monitoring' := 'call'}
PROPERTY ErrorId : UDINT
GET
ErrorId := MCReset.ErrorID;
END_GET
END_PROPERTY

METHOD Execute : BOOL
IF _Axis.Axis.Status.Coupled AND NOT _Axis.Axis.Status.Error THEN
	Execute := TRUE;
	RETURN;
ELSIF Busy OR _Axis.Axis.Status.Coupled THEN
	Execute := TRUE;
	RETURN;
END_IF

SequenceState := 10;
Execute		  := TRUE;
END_METHOD

END_FUNCTION_BLOCK

// ---- _Internal/MotionTasks/MC2/Reset/Mc2SoEResetTask.TcPOU
FUNCTION_BLOCK Mc2SoEResetTask EXTENDS Mc2MotionTask
VAR
	MCReset		  : Tc2_MC2.MC_Reset;
	SoEReset	  : FB_SoEReset;
	SequenceState : UDINT;
	_ErrorId	  : UDINT;
END_VAR

{attribute 'monitoring' := 'call'}
PROPERTY Busy : BOOL
GET
Busy := SequenceState <> 0;
END_GET
END_PROPERTY

METHOD CyclicLogic
VAR_INST
	ResetDelay : TON;
END_VAR
CASE SequenceState OF
	0: // Wait for Execute()
	10:
		SoEReset.Execute := TRUE;
		SequenceState	 := SequenceState + 10;

	20:
		IF NOT SoEReset.Busy THEN
			IF SoEReset.Error THEN
				IF SoEReset.SercosErrId < 0 THEN
					_ErrorID := SoEReset.SercosErrId;
				ELSE
					_ErrorID := SoEReset.AdsErrId;
				END_IF

				SequenceState := 999;
			ELSE
				//No error occurred
				SequenceState := SequenceState + 10;
			END_IF
		END_IF

	30:
		MCReset.Execute := TRUE;
		SequenceState	:= SequenceState + 10;

	40:
		IF NOT MCReset.Busy THEN
			SequenceState := SequenceState + 10;
		END_IF

	50:
		ResetDelay(IN := TRUE);
		IF ResetDelay.Q OR NOT _Axis.Axis.Status.DriveDeviceError THEN
			ResetDelay(IN := FALSE);
			SequenceState := 0;
		END_IF

	999:
		_ErrorId	  := 0;
		SequenceState := 0;
END_CASE

SoEReset(Axis := _Axis.Axis);
MCReset(Axis := _Axis.Axis);
SoEReset.Execute := FALSE;
MCReset.Execute	 := FALSE;
END_METHOD

{attribute 'monitoring' := 'call'}
PROPERTY Error : BOOL
GET
Error := SequenceState = 999;
END_GET
END_PROPERTY

{attribute 'monitoring' := 'call'}
PROPERTY ErrorId : UDINT
GET
ErrorId := _ErrorID;
END_GET
END_PROPERTY

METHOD Execute : BOOL
IF _Axis.Axis.Status.Coupled AND NOT _Axis.Axis.Status.Error THEN
	Execute := TRUE;
	RETURN;
ELSIF Busy OR _Axis.Axis.Status.Coupled THEN
	Execute := TRUE;
	RETURN;
END_IF

SequenceState := 10;
Execute		  := TRUE;
END_METHOD

END_FUNCTION_BLOCK

// ---- _Internal/MotionTasks/MC3/Home/Mc3MotionHomeTask_SetPosition.TcPOU
FUNCTION_BLOCK Mc3MotionHomeTask_SetPosition EXTENDS Mc3MotionTask
VAR
	MCSetPosition : Tc3_Mc3Ptp.MC_SetPosition;
	_HomePosition : LREAL := 0.0;
END_VAR

{attribute 'monitoring' := 'call'}
PROPERTY Busy : BOOL
GET
Busy := MCSetPosition.Busy;
END_GET
END_PROPERTY

METHOD CyclicLogic
MCSetPosition(Axis := _Axis.Axis, Position := HomePosition);
MCSetPosition.Execute := FALSE;
END_METHOD

{attribute 'monitoring' := 'call'}
PROPERTY Error : BOOL
GET
Error := MCSetPosition.Error;
END_GET
END_PROPERTY

{attribute 'monitoring' := 'call'}
PROPERTY ErrorId : UDINT
GET
ErrorId := MCSetPosition.ErrorID;
END_GET
END_PROPERTY

METHOD Execute : BOOL
IF Axis.Busy OR Axis.Error THEN
	RETURN;
END_IF

MCSetPosition.Execute := TRUE;
Execute				  := TRUE;
END_METHOD

PROPERTY HomePosition : LREAL
GET
HomePosition := MCSetPosition.Position;
END_GET
SET
MCSetPosition.Position := HomePosition;
END_SET
END_PROPERTY

END_FUNCTION_BLOCK

// ---- _Internal/MotionTasks/MC3/Home/Mc3MotionHomeTask_SetZeroHere.TcPOU
FUNCTION_BLOCK Mc3MotionHomeTask_SetZeroHere EXTENDS Mc3MotionTask
VAR
	MCSetPosition : Tc3_Mc3Ptp.MC_SetPosition;
END_VAR

{attribute 'monitoring' := 'call'}
PROPERTY Busy : BOOL
GET
Busy := MCSetPosition.Busy;
END_GET
END_PROPERTY

METHOD CyclicLogic
MCSetPosition(Axis := _Axis.Axis);
MCSetPosition.Execute := FALSE;
END_METHOD

{attribute 'monitoring' := 'call'}
PROPERTY Error : BOOL
GET
Error := MCSetPosition.Error;
END_GET
END_PROPERTY

{attribute 'monitoring' := 'call'}
PROPERTY ErrorId : UDINT
GET
ErrorId := MCSetPosition.ErrorID;
END_GET
END_PROPERTY

METHOD Execute : BOOL
IF Axis.Busy OR Axis.Error THEN
	RETURN;
END_IF

MCSetPosition.Execute := TRUE;
Execute				  := TRUE;
END_METHOD

END_FUNCTION_BLOCK

// ---- _Internal/MotionTasks/MC3/Power/Mc3StopTask.TcPOU
FUNCTION_BLOCK Mc3StopTask EXTENDS Mc3MotionTask IMPLEMENTS I_Mc3MotionTask
VAR
	McHalt : Tc3_Mc3Ptp.MC_Halt;
END_VAR

{attribute 'monitoring' := 'call'}
PROPERTY Busy : BOOL
GET
Busy := McHalt.Busy;
END_GET
END_PROPERTY

METHOD CyclicLogic
McHalt(Axis			  := _Axis.Axis,
	   Deceleration	  := _Axis.Deceleration,
	   Jerk			  := _Axis.Jerk,
	   Done			  =>,
	   Busy			  =>,
	   Active		  =>,
	   CommandAborted =>,
	   Error		  =>,
	   ErrorId		  =>);

McHalt.Execute := FALSE;
END_METHOD

{attribute 'monitoring' := 'call'}
PROPERTY Error : BOOL
GET
Error := McHalt.Error;
END_GET
END_PROPERTY

{attribute 'monitoring' := 'call'}
PROPERTY ErrorId : UDINT
GET
ErrorId := McHalt.ErrorID;
END_GET
END_PROPERTY

METHOD Execute : BOOL
McHalt(Axis			:= _Axis.Axis,
	   Execute		:= TRUE,
	   Deceleration := _Axis.Deceleration,
	   Jerk			:= _Axis.Jerk);

Execute := TRUE;
END_METHOD

END_FUNCTION_BLOCK

// ---- _Internal/MotionTasks/MC3/Reset/Mc3CoEResetTask.TcPOU
FUNCTION_BLOCK Mc3CoEResetTask EXTENDS Mc3MotionTask
VAR
	MCReset		  : Tc3_Mc3Ptp.MC_Reset;
	SequenceState : UDINT;
END_VAR

{attribute 'monitoring' := 'call'}
PROPERTY Busy : BOOL
GET
Busy := SequenceState <> 0;
END_GET
END_PROPERTY

METHOD CyclicLogic
CASE SequenceState OF
	0: // Wait for Execute()
	10:
		MCReset.Execute := TRUE;
		SequenceState	:= SequenceState + 10;

	20:
		IF NOT MCReset.Busy THEN
			SequenceState := 0;
		END_IF
END_CASE

MCReset(Axis := _Axis.Axis);
MCReset.Execute := FALSE;
END_METHOD

{attribute 'monitoring' := 'call'}
PROPERTY Error : BOOL
GET
Error := MCReset.Error;
END_GET
END_PROPERTY

{attribute 'monitoring' := 'call'}
PROPERTY ErrorId : UDINT
GET
ErrorId := MCReset.ErrorID;
END_GET
END_PROPERTY

METHOD Execute : BOOL
VAR
    Coupled : BOOL;
END_VAR
Coupled := _Axis.Axis.McToPlc.Std.AxisState = EAxisState.SynchronizedMotion;
IF Coupled AND NOT _Axis.Axis.McToPlc.Std.HasError THEN
	Execute := TRUE;
	RETURN;
ELSIF Busy OR Coupled THEN
	Execute := TRUE;
	RETURN;
END_IF

SequenceState := 10;
Execute		  := TRUE;
END_METHOD

END_FUNCTION_BLOCK

// ---- _Internal/Tracing/LocalLogger.TcPOU
FUNCTION_BLOCK LocalLogger
VAR_GENERIC CONSTANT
	LogSize : UDINT := 5;
END_VAR IMPLEMENTS I_TraceLogger
VAR
	_Messages : ARRAY[0..LogSize - 1] OF T_MaxString;
END_VAR

METHOD ClearLog
VAR_INPUT
END_VAR
VAR
	i : UDINT;
END_VAR
FOR i := 0 TO LogSize - 1 DO
	_Messages[i] := '';
END_FOR
END_METHOD

METHOD LogMessage
VAR_INPUT
	Key		  : T_MaxString;
	Value	  : T_MaxString;
	SourceId  : UDINT := 0;
	TimeStamp : ULINT := 0;
	MessageId : UDINT := 1;
	Severity  : USINT := 1;
END_VAR

VAR
	_TimeStamp  : T_FILETIME64;
	TimeString : T_MaxString;
	i : UDINT;
END_VAR
IF TimeStamp = 0 THEN
	_TimeStamp := F_GetSystemTime();
ELSE
	_TimeStamp := Timestamp;
END_IF

TimeString := SYSTEMTIME_TO_STRING(FILETIME64_TO_SYSTEMTIME(_TimeStamp));
//shift messages down
FOR i := 1 TO LogSize - 1 DO
	_Messages[LogSize - i] := _Messages[LogSize - 1 - i];
END_FOR

_Messages[0] := CONCAT(TimeString, CONCAT(' ', CONCAT(Key, CONCAT('- Sev:', CONCAT(TO_STRING(Severity), CONCAT(' ', CONCAT(Key, CONCAT(': ', Value))))))));
END_METHOD

{attribute 'monitoring' := 'call'}
PROPERTY Messages : REFERENCE TO ARRAY[0..LogSize - 1] OF T_MaxString
GET
Messages REF= _Messages;
END_GET
END_PROPERTY

END_FUNCTION_BLOCK

// ---- _Internal/Tracing/TraceMessageInfo.TcPOU
{attribute 'hide_all_locals'}
FUNCTION_BLOCK TraceMessageInfo IMPLEMENTS I_TraceMessageInfo
VAR
	_Message   : T_MaxString;
	_MessageId : UDINT;
	_Severity  : USINT;
END_VAR

{attribute 'monitoring':='call'}
PROPERTY Message : T_MaxString
GET
Message := _Message;
END_GET
SET
_Message := Message;
END_SET
END_PROPERTY

{attribute 'monitoring':='call'}
PROPERTY MessageId : UDINT
GET
MessageId := _MessageId;
END_GET
SET
_MessageId := MessageId;
END_SET
END_PROPERTY

{attribute 'monitoring':='call'}
PROPERTY Severity : USINT
GET
Severity := _Severity;
END_GET
SET
_Severity := Severity;
END_SET
END_PROPERTY

END_FUNCTION_BLOCK

// ---- _Internal/Tracing/TraceSourceInfo.TcPOU
{attribute 'hide_all_locals'}
FUNCTION_BLOCK TraceSourceInfo IMPLEMENTS I_TraceSourceInfo
VAR
	_SourceId	: UDINT;
	_SourceName : T_MaxString;
	_TimeStamp	: ULINT;
END_VAR

{attribute 'monitoring' := 'call'}
PROPERTY SourceId : UDINT
GET
SourceId := _SourceId;
END_GET
SET
_SourceId := SourceId;
END_SET
END_PROPERTY

{attribute 'monitoring' := 'call'}
PROPERTY SourceName : T_MaxString
GET
SourceName := _SourceName;
END_GET
SET
_SourceName := SourceName;
END_SET
END_PROPERTY

{attribute 'monitoring' := 'call'}
PROPERTY TimeStamp : ULINT
GET
TimeStamp := _TimeStamp;
END_GET
SET
_TimeStamp := TimeStamp;
END_SET
END_PROPERTY

END_FUNCTION_BLOCK
